# EPICS autosave request: iocBoot/gmca_23i_ioc2/dbSave/digital_IO_16_desc.req
%
% This request file stores settings for Acromag 9440 digital out
%

$(P)0.DESC
$(P)1.DESC
$(P)2.DESC
$(P)3.DESC
$(P)4.DESC
$(P)5.DESC
$(P)6.DESC
$(P)7.DESC
$(P)8.DESC
$(P)9.DESC
$(P)10.DESC
$(P)11.DESC
$(P)12.DESC
$(P)13.DESC
$(P)14.DESC
$(P)15.DESC
